Fanuc KAREL source: compact_preamble.KL

PROGRAM KD00021
%NOLOCKGROUP
VAR
I:INTEGER;J:INTEGER;B:BOOLEAN;R:REAL;S : STRING[80]
EXTVAL FROM KD00001 : INTEGER
BEGIN
I=EXTVAL
END KD00021
